{attribute 'linkalways'} 
{attribute 'no_explicit_call' := 'This FB is a CLASS and must be accessed using methods or properties'}
{attribute 'enable_dynamic_creation'}
FUNCTION_BLOCK _LWORD EXTENDS DatatypeBase
VAR
	localData : LWORD;
	activeData : REFERENCE TO LWORD REF= localData;
END_VAR

PROPERTY PUBLIC Address : PVOID
GET
Address := ADR(activeData);
END_GET
END_PROPERTY

METHOD PUBLIC ClearReference
VAR_INPUT
END_VAR
activeData REF= localData;
END_METHOD

METHOD PUBLIC Clone : I_Datatype
VAR
    pClone : POINTER TO _LWORD;
END_VAR
pClone := __NEW(_LWORD(InitialValue := Value));
Clone := pClone^;
END_METHOD

METHOD FB_init : BOOL
VAR_INPUT
	bInitRetains : BOOL; // if TRUE, the retain variables are initialized (warm start / cold start)
	bInCopyCode : BOOL;  // if TRUE, the instance afterwards gets moved WORDo the copy code (online change)
	InitialValue : LWORD;
END_VAR
localData := InitialValue;
END_METHOD

PROPERTY PUBLIC IecType : T_MAXSTRING
GET
IecType := 'LWORD';
END_GET
END_PROPERTY

METHOD PUBLIC MakeReferenceTo
VAR_INPUT
	ReferenceTarget : REFERENCE TO LWORD;
END_VAR
activeData REF= ReferenceTarget;
END_METHOD

METHOD PUBLIC SerializeWith
VAR_INPUT
	Serializer : I_Serializer;
END_VAR
Serializer.AddLword(activeData);
END_METHOD

PROPERTY PUBLIC Size : UDINT
GET
Size := SIZEOF(activeData);
END_GET
END_PROPERTY

METHOD TryDeserializeFrom : BOOL
VAR_INPUT
	Deserializer : I_Deserializer;
END_VAR
TryDeserializeFrom := Deserializer.TryGetLword(activeData);
END_METHOD

METHOD TryMakeReferenceTo : BOOL
VAR_INPUT
	Target : I_Datatype;
END_VAR
VAR
	pTargetData : POINTER TO LWORD;
END_VAR
IF NOT (Target.IecType = IecType) THEN
	RETURN;
END_IF

pTargetData := Target.Address;
activeData REF= pTargetData^;
TryMakeReferenceTo := TRUE;
END_METHOD

PROPERTY PUBLIC Value : LWORD
GET
Value := activeData;
END_GET
SET
activeData := Value;
END_SET
END_PROPERTY

END_FUNCTION_BLOCK

(* stored: Version 1.1.0.1, ProductVersion 3.1.4024.12
   POU _LWORD: Id {83eb2057-61c3-0f5c-2bbd-2c1a0c4bcdbb}, SpecialFunc None
   Folder Constructor: Id {76a599ac-f355-0c91-3411-2c4573633eb2}
   Property Address: Id {3ea38e9d-e5b4-08f8-3bac-d50de01d8088}
   Get Get: Id {4c3c2f62-1325-05ee-2e66-2b5f5411ac84}
   Method ClearReference: Id {10b74754-dd3d-0784-2dc0-bc9aaaa6dff2}
   Method Clone: Id {70ec616f-2c61-064a-2209-68affc8cda70}
   Method FB_init: Id {6fbd1526-f642-03c9-1957-3df80912e78f}
   Property IecType: Id {f1ea044d-8243-0a57-0c7e-1f8798251cf8}
   Get Get: Id {7c6d7a65-de1e-06bb-2224-776a3f729bc6}
   Method MakeReferenceTo: Id {22dc0f3b-b797-03c0-006f-7c61fb3682bc}
   Method SerializeWith: Id {43957286-f88e-05ee-30ce-fc0a753ce5f1}
   Property Size: Id {e6a57ecf-e117-0957-19ab-e82010e77df9}
   Get Get: Id {e9dcdc74-ac46-04bd-0982-1d0e341f3ca2}
   Method TryDeserializeFrom: Id {0e99a354-8f0e-0ad8-03af-ecb45be70e2a}
   Method TryMakeReferenceTo: Id {7534ac8b-b439-087c-0eca-0e1f7561613f}
   Property Value: Id {32408784-0d34-0b64-3e25-e04ead8e7528}
   Get Get: Id {4b97d08e-c899-0a71-3b3b-f66d8e13a09d}
   Set Set: Id {4a2d1657-4af8-0535-24f3-4c03181dcf25} *)
